PROGRAM POU_DALI_Prog_Final
VAR
    fbRecallMax : Tc3_DALI.FB_DALI102RecallMaxLevel(POU_Comm.fbKL6821Communication);
    fbOff       : Tc3_DALI.FB_DALI102Off(POU_Comm.fbKL6821Communication);
END_VAR

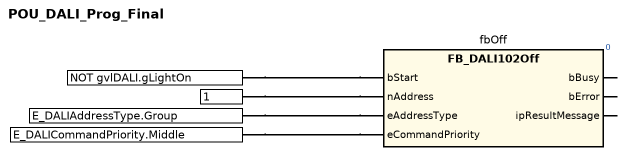
fbOff(
    bStart := NOT gvlDALI.gLightOn,
    nAddress := 1,
    eAddressType := E_DALIAddressType.Group,
    eCommandPriority := E_DALICommandPriority.Middle); // FB_DALI102Off

END_PROGRAM

(* stored: Version 1.1.0.1, ProductVersion 3.1.4024.15
   POU POU_DALI_Prog_Final: Id {e1e63b0b-1b77-4d24-a7d4-2bfb10d77c35}, SpecialFunc None *)
